TYPE ST_ui_control :
STRUCT
	draping_enable:BOOL; //台车自动摆位---姿态调整为建立无菌屏障时所需状态--结束后给定结束信号
	docking_enable:BOOL; //台车自动摆位---姿态调整为进入无菌区时所需状态（器械对接姿态）--结束后给定结束信号
	stow_enable:BOOL; //所有机械臂收纳使能
	joysticks_enable:BOOL; //通过手柄按钮，任意拖动机械臂所有关节
	camera_joysticks_enable:BOOL;//相机界面中的使能按钮
	limit_height_adjusting:BOOL; //限制高度调整，true:使能，false:禁止
END_STRUCT
END_TYPE

(* stored: Version 1.1.0.1, ProductVersion 3.1.4024.11
   DUT ST_ui_control: Id {5feec175-de79-40fc-b60d-eb6c37040d35} *)
